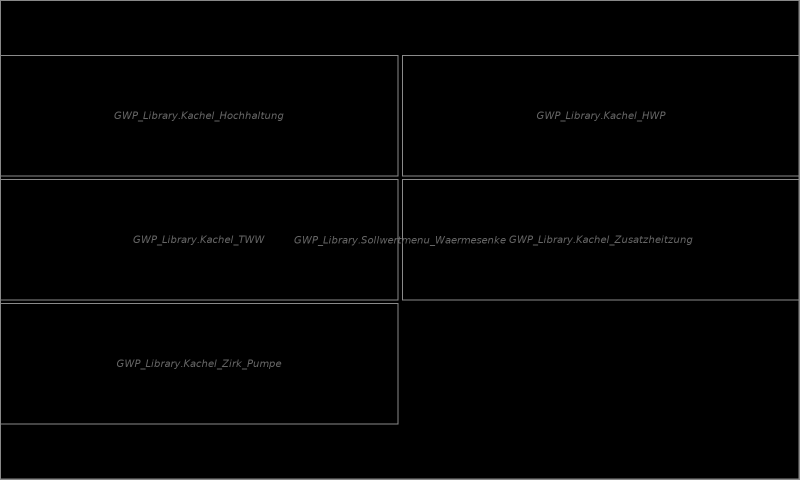
VISUALIZATION Sollwertmenu_Waermesenke  // 800x480
    Frame (0,55 398x121)
        shows GWP_Library.Kachel_Hochhaltung()
        OnMouseClick: change screen: Sollwertmenu_KD
    Frame (402,55 398x121)
        shows GWP_Library.Kachel_HWP()
        OnMouseClick: change screen: Sollwertmenu_HWP
    Frame (0,179 398x121)
        shows GWP_Library.Kachel_TWW()
        OnMouseClick: change screen: Sollwertmenu_TWW
    Frame (402,179 398x121)
        shows GWP_Library.Kachel_Zusatzheitzung()
        OnMouseClick: change screen: Zusatzheizung_Sollwerte
    Frame (0,303 398x121)
        shows GWP_Library.Kachel_Zirk_Pumpe()
        OnMouseClick: change screen: Sollwertmenu_Zirk_PU
    Frame (0,0 800x480)
        shows GWP_Library.Sollwertmenu_Waermesenke(FB_Init_1 := Main.Init_0)
END_VISUALIZATION

(* stored: Version 1.1.0.1, ProductVersion 3.1.4022.6
   Visu Sollwertmenu_Waermesenke: Id {ad908f14-0f60-4945-9739-da53893af235} *)
